Staubli VAL3: getFieldValue.pgx

public program getFieldValue(string x_sCaption, string& x_sValue[], num x_nError)
  local num l_i
  local bool l_bFound
  local bool l_bQuit
begin
  // This program returns the value of the field passed as parameter
  //
  // Input Param
  //  x_sCaption      : Name of the field
  //
  // Output Param
  //  x_sValue      : Current value
  //  x_nError      : Error code
  //                = 0 success
  //                = 1 Caption  not found
  //Created 21/12/05                              CCUR
  //--------------------------------------------------------------
  x_nError=0
  // Search if label passed as parameter is known
  l_i=0
  do
    l_bFound=(x_sCaption==pw:sTxtBoxCaption[l_i])
    l_i=l_i+1
  until (l_bFound or (l_i>=nNumOfTxtBox))
  //
  if l_bFound
    x_sValue=pw:sTxtBoxVal[l_i-1]
  else
    x_nError=4
    // Prepare clear text error message
    call ut:addStrToString(sErrMsgList[x_nError],sErrorMessage,"",x_sCaption)
  endIf
end
